TYPE ST_Value :
STRUCT
	Setpoint	: T_ControllerValue;
	Actual		: T_ControllerValue;
END_STRUCT
END_TYPE

(* stored: Version 1.1.0.1, ProductVersion 3.1.4024.14
   DUT ST_Value: Id {13cd15ac-5031-0740-27bc-f970d26ec4ee} *)
